// TIA Portal V17 export
// export: Created 2025-03-05T08:02:24.459736Z, ExportSetting WithDefaults, DisplayName Totally Integrated Automation Portal, DisplayVersion V17 Update 8, DisplayName TIA Portal Openness, DisplayVersion V17 Update 8, DisplayName TIA Portal Version Control Interface, DisplayVersion V17, DisplayName SINAMICS Startdrive Advanced, DisplayVersion V17 SP2, DisplayName SINAMICS Startdrive G110M, G120, G120C, G120D, G120P, G115D, DisplayVersion V17 SP2, DisplayName SINAMICS Startdrive G130, G150, S120, S150, SINAMICS MV, S210, DisplayVersion V17 SP2, DisplayName STEP 7 Professional, DisplayVersion V17 Update 8, DisplayName SINUMERIK ONE STEP 7 Toolbox, DisplayVersion V17 Update 12, DisplayName SINUMERIK 840D sl STEP 7 Toolbox, DisplayVersion V17 Update 12, DisplayName STEP 7 Safety, DisplayVersion V17 Update 6, DisplayName WinCC Advanced, DisplayVersion V17 Update 8
TYPE "INTERLOCKS_ETXETAR_ROBOT_CELL_PER_UNIT"
// stored: IsFailsafeCompliant false
   STRUCT
      MACHINE_TO_ROBOT : Struct
         MCH_HEARTBEAT : Bool;   // MACHINE HEARTBEAT (MACHINE TO GANTRY) / MACHINE HEARTBEAT
         MCH_E_STOP_OK : Bool;   // MACHINE EMERGENCY STOP OK (MACHINE TO GANTRY) / MACHINE EMERGENCY STOP OK
         MCH_FAULT : Bool;   // MACHINE FAULT PRESENT
         MCH_SAFETY_DOORS_CLSD_LCKD : Bool;   // MACHINE SAFETY GATES OK (LOCKED)(MACHINE TO GANTRY) / MACHINE SAFETY DOORS CLOSED AND LOCKED
         SPARE_0_4 : Bool;
         SPARE_0_5 : Bool;
         MCH_MANUAL_MODE : Bool;   // MACHINE IN MANUAL MODE (MACHINE TO GANTRY) / MACHINE MANUAL MODE SELECTED
         MCH_AUTO_MODE : Bool;   // MACHINE IN AUTO MODE(MACHINE TO GANTRY) / MACHINE AUTO MODE SELECTED
         MCH_AUTO_CYCLE_RUN : Bool;   // MACHINE AUTO CYCLE RUNNING (MACHINE TO GANTRY) / MACHINE CYCLE RUNNING IN AUTOMATIC MODE
         MCH_WARM_UP_CYCLE_RUN : Bool;   // MACHINE IS IN WARMUP CYCLE (MACHINE TO GANTRY) / MACHINE WARM UP CYCLE RUNNING
         MCH_RUN_OUT_CYCLE : Bool;   // MACHINE IN RUN OUT MODE (MACHINE TO GANTRY) / MACHINE RUN OUT CYCLE SELECTED
         MCH_CALIBRATION_CYCLE : Bool;   // MACHINE CALIBRATION CYCLE SELECTED
         MCH_MASTER_MEASUREMENT_CYCLE : Bool;   // MACHINE MASTER MEASUREMENT CYCLE SELECTED
         MCH_PART_DEMAND_SOON : Bool;   // MACHINE PART DEMAND SOON (MACHINE TO GANTRY) / MACHINE PART DEMAND SOON
         MCH_SAFETY_DOOR_OPEN_REQ : Bool;   // MACHINE SAFETY DOOR OPEN REQUEST
         MCH_CELL_SAFETY_DOOR_OK_TO_OPEN : Bool;   // MACHINE APPROVAL TO OPEN THE CELL SAFETY DOOR
         MCH_EMPTY : Bool;   // MACHINE EMPTY
         MCH_FIX_1_ENABLED : Bool;   // MACHINE FIXTURE 1 ENABLED FOR LOAD/UNLOAD
         MCH_FIX_2_ENABLED : Bool;   // MACHINE FIXTURE 2 ENABLED FOR LOAD/UNLOAD
         MCH_FIX_3_ENABLED : Bool;   // MACHINE FIXTURE 3 ENABLED FOR LOAD/UNLOAD
         MCH_FIX_4_ENABLED : Bool;   // MACHINE FIXTURE 4 ENABLED FOR LOAD/UNLOAD
         MCH_FIX_1_PART_PRSNT : Bool;   // MACHINE FIXTURE 1 PART PRESENT
         MCH_FIX_2_PART_PRSNT : Bool;   // MACHINE FIXTURE 2 PART PRESENT
         MCH_FIX_3_PART_PRSNT : Bool;   // MACHINE FIXTURE 3 PART PRESENT
         MCH_FIX_4_PART_PRSNT : Bool;   // MACHINE FIXTURE 4 PART PRESENT
         MCH_FIX_1_CALIBRATION_REQ : Bool;   // MACHINE FIXTURE 1 CALIBRATION REQUIRED
         MCH_FIX_2_CALIBRATION_REQ : Bool;   // MACHINE FIXTURE 2 CALIBRATION REQUIRED
         MCH_FIX_3_CALIBRATION_REQ : Bool;   // MACHINE FIXTURE 3 CALIBRATION REQUIRED
         MCH_FIX_4_CALIBRATION_REQ : Bool;   // MACHINE FIXTURE 4 CALIBRATION REQUIRED
         SPARE_3_5 : Bool;
         SPARE_3_6 : Bool;
         SPARE_3_7 : Bool;
         CLEAR_LOAD_UNLOAD : Bool;   // MACHINE PART TYPE CHANGE IS POSSIBLE (MACHINE TO GANTRY) / MACHINE CLEAR TO LOAD / UNLOAD PARTS
         MCH_UNLOAD_REQUEST_FACE_R : Bool;   // MACHINE UNLOAD REQUEST FACE R
         MCH_UNLOAD_REQUEST_FACE_N : Bool;   // MACHINE UNLOAD REQUEST FACE N
         MCH_LOAD_REQUEST_FACE_R : Bool;   // MACHINE LOAD REQUEST FACE R
         MCH_LOAD_REQUEST_FACE_N : Bool;   // MACHINE SUSPECT PART FROM MACHINE (MACHINE TO GANTRY) / MACHINE LOAD REQUEST FACE N
         MCH_UNLD_ANTICIPATION_FACE_R : Bool;   // MACHINE EMPTY (MACHINE TO GANTRY) / MACHINE UNLOAD ANTICIPATION FACE R
         MCH_UNLD_ANTICIPATION_FACE_N : Bool;   // MACHINE UNLOAD ANTICIPATION FACE N
         MCH_LOAD_ANTICIPATION_FACE_R : Bool;   // MACHINE QUALITY CHECK WARNING (MACHINE TO GANTRY) / MACHINE LOAD ANTICIPATION FACE R
         MCH_LOAD_ANTICIPATION_FACE_N : Bool;   // MACHINE QUALITY CHECK FAULT (MACHINE TO GANTRY) / MACHINE LOAD ANTICIPATION FACE N
         MCH_PART_A_PRESENT : Bool;   // MACHINE QUALITY CHECK FAULT (MACHINE TO GANTRY) / MACHINE PART A PRESETN
         MCH_PART_A_MACHINED : Bool;   // MACHINE QUALITY CHECK FAULT (MACHINE TO GANTRY) / MACHINE PART A MACHINED
         MCH_PART_A_REJECTED : Bool;   // MACHINE QUALITY CHECK ACKNOWLEDGED (MACHINE TO GANTRY) / MACHINE PART A REJECTED
         MCH_PART_A_QUALITY : Bool;   // MACHINE PART A QUALITY
         SPARE_5_5 : Bool;   // MACHINE READY TO ACCEPT REWORK PART (MACHINE TO GANTRY)
         SPARE_5_6 : Bool;
         SPARE_5_7 : Bool;
         SPARE_6_0 : Bool;   // MACHINE CLEAR TO LOAD/UNLOAD (MACHINE TO GANTRY)
         SPARE_6_1 : Bool;   // MACHINE READY TO UNLOAD PART (MACHINE TO GANTRY)
         SPARE_6_2 : Bool;   // MACHINE READY TO LOAD PART (MACHINE TO GANTRY)
         SPARE_6_3 : Bool;   // MACHINE PART PRESENT (MACHINE TO GANTRY)
         SPARE_6_4 : Bool;   // MACHINE GOOD PART (MACHINE TO GANTRY)
         SPARE_6_5 : Bool;
         SPARE_6_6 : Bool;
         SPARE_6_7 : Bool;
         MCH_PART_TYPE : Byte;   // MACHINE PART IS CLAMPED (MACHINE TO GANTRY) / MACHINE PART TYPE
         SPARE : Array[0..55] of Byte;
      END_STRUCT;
      ROBOT_TO_MACHINE : Struct
         RBT_HEARTBEAT : Bool;   // GANTRY HEARTBEAT (GANTRY TO MACHINE) / ROBOT HEARTBEAT
         RBT_E_STOP_OK : Bool;   // GANTRY EMERGENCY STOP OK (GANTRY TO MACHINE) / ROBOT EMERGENCY STOP OK
         RBT_FAULT : Bool;   // ROBOT FAULT PRESENT
         RBT_SAFETY_DOOR_CLSD_LCKD : Bool;   // ROBOT SAFETY DOOR CLOSED AND LOCKED
         RBT_CELL_EMPTY : Bool;   // ROBOT CELL EMPTY
         SPARE_0_5 : Bool;
         SPARE_0_6 : Bool;
         SPARE_0_7 : Bool;
         RBT_MANUAL_MODE : Bool;   // GANTRY IN MANUAL MODE (GANTRY TO MACHINE) / ROBOT MANUAL MODE SELECTED
         RBT_AUTO_MODE : Bool;   // GANTRY IN AUTO MODE (GANTRY TO MACHINE) / ROBOT AUTO MODE SELECTED
         RBT_AUTO_CYCLE_RUN : Bool;   // GANTRY IN AUTO CYCLE RUNNING (GANTRY TO MACHINE) / ROBOT CYCLE RUNNING IN AUTOMATIC MODE
         SPARE_1_3 : Bool;   // GANTRY OVERHEAD DOOR CLOSED & LOCKED (GANTRY TO MACHINE)
         RBT_RUN_OUT_REQ : Bool;   // GANTRY PART TYPE CHANGE REQUESTED (GANTRY TO MACHINE) / ROBOT MACHINE RUN OUT REQUEST
         RBT_RUN_OUT_COMPLETED : Bool;   // GANTRY IN RUN OUT COMPLETE(GANTRY TO MACHINE) / ROBOT RUN OUT COMPLETED
         RBT_SAFETY_DOOR_OPEN_REQ : Bool;   // ROBOT ANY CELL SAFETY DOOR OPEN REQUEST
         RBT_MCH_SAFETY_DOOR_OK_TO_OPEN : Bool;   // ROBOT APPROVAL TO OPEN THE MACHINE SAFETY DOOR
         RBT_READY_TO_SERVICE : Bool;   // ROBOT IS READY TO SERVICE THE MACHINE
         RBT_OUT_OF_COLLISION_MACHINE : Bool;   // GANTRY CLEAR OF MACHINE (GANTRY TO MACHINE) / ROBOT OUT OF COLLISION MACHINE
         RBT_OUT_OF_COLLISION_FIXTURE : Bool;   // GANTRY CLEAR OF FIXTURE (GANTRY TO MACHINE) / ROBOT OUT OF COLLISION FIXTURE
         SPARE_2_3 : Bool;
         SPARE_2_4 : Bool;
         SPARE_2_5 : Bool;
         SPARE_2_6 : Bool;
         SPARE_2_7 : Bool;
         SPARE_3_0 : Bool;
         SPARE_3_1 : Bool;
         SPARE_3_2 : Bool;
         SPARE_3_3 : Bool;
         SPARE_3_4 : Bool;
         SPARE_3_5 : Bool;
         SPARE_3_6 : Bool;
         SPARE_3_7 : Bool;
         RBT_PART_ENABLED : Bool;   // ROBOT PART ENABLED
         SPARE_4_1 : Bool;   // GANTRY READY TO SERVICE MACHINE (GANTRY TO MACHINE)
         RBT_PART_FACE_R_TO_DELIVER : Bool;   // ROBOT PART FACE R TO DELIVER IMMEDIATELY
         RBT_PART_FACE_N_TO_DELIVER : Bool;   // ROBOT PART FACE N TO DELIVER IMMEDIATELY
         RBT_OUT_OF_PARTS_FACE_R_TO_DELIVER : Bool;   // ROBOT OUT OF PARTS FACE R IN CELL TO DELIVER
         RBT_OUT_OF_PARTS_FACE_N_TO_DELIVER : Bool;   // ROBOT OUT OF PARTS FACE N IN CELL TO DELIVER
         SPARE_4_6 : Bool;
         SPARE_4_7 : Bool;
         RBT_PART_LOADED : Bool;   // ROBOT PART LOADED
         RBT_PART_UNLOADED : Bool;   // ROBOT PART UNLOADED
         SPARE_5_2 : Bool;
         SPARE_5_3 : Bool;
         RBT_FIX_SKIP_REQ : Bool;   // ROBOT FIXTURE SKIP REQUEST
         SPARE_5_5 : Bool;
         SPARE_5_6 : Bool;
         SPARE_5_7 : Bool;
         RBT_PART_TYPE_REQ : Bool;   // ROBOT PART TYPE CHANGE REQUEST
         SPARE_6_1 : Bool;
         SPARE_6_2 : Bool;
         SPARE_6_3 : Bool;
         SPARE_6_4 : Bool;   // GANTRY ROUGH PART IS REWORK PART (GANTRY TO MACHINE)
         SPARE_6_5 : Bool;
         SPARE_6_6 : Bool;
         SPARE_6_7 : Bool;
         RBT_PART_TYPE : Byte;   // ROBOT PART TYPE
         SPARE : Array[0..55] of Byte;
      END_STRUCT;
   END_STRUCT;
END_TYPE
